PROGRAM DP_CONFIG_OUT_EL6731
VAR
END_VAR

DP_MISO_WORD_1:=SET_NC_PARAM_1;	
DP_MISO_WORD_2:=SET_NC_PARAM_2;
DP_MISO_WORD_3:=SET_NC_PARAM_3;													
DP_MISO_WORD_4:=SET_NC_PARAM_4;

END_PROGRAM

(* stored: Version 1.1.0.1, ProductVersion 3.1.0.26
   POU DP_CONFIG_OUT_EL6731: Id {f39ae699-8486-4bf9-afa7-fc8bcd4e59d7} *)
